FUNCTION_BLOCK STEST_END (* Service Interface Function Block Type *)
  (* Description: Copyright (c) 2015 Profactor GmbH This program and the accompanying materials are made available under the terms of the Eclipse Public License 2.0 which is available at https://www.eclipse.org/legal/epl-2.0/ SPDX-License-Identifier: EPL-2.0 *)
  (* Version 3.0, 2025-04-14, Patrick Aigner, changed package *)
  (* Version 1.0, 2015-01-11, Michael Hofmann, Profactor GmbH *)
  PACKAGE eclipse4diac::utils;
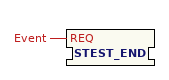
  EVENT_INPUT
    REQ; (* Service Request *)
  END_EVENT
END_FUNCTION_BLOCK
